TYPE ST_ManualModeStatus :
STRUCT
    eState                     : E_ManualModeState;
    eMessage                   : E_ManualModeMessage;
    bActive                    : BOOL;
    bSafeToExit                : BOOL;
    bIndexPermissive           : BOOL;
    bAssemblySupportPermissive : BOOL; 
    bSiliconeSupportPermissive : BOOL;
    bDoorUnlockPermissive      : BOOL;
    bEquipmentStartPermissive  : BOOL;
	// IVEK Prime
	bIvekPrimePermissive 		: BOOL;

    // Manual Assembly / Flipping Station
    bAssemblyStationStartPermissive : BOOL;

    bCommandRejected           : BOOL;
    sMessage                   : STRING(255);
	

    // Manual Silicone Station
    bSiliconeStationStartPermissive     : BOOL;

END_STRUCT
END_TYPE

(* stored: Version 1.1.0.1, ProductVersion 3.1.4026.18
   DUT ST_ManualModeStatus: Id {69e8599d-00b6-491b-94f6-86fee5a77320} *)
